(* PLC project liner_cyclic.project, CODESYS CODESYS V3.5 SP17 Patch 3 *)
(* stored: creationDateTime 1970-01-01T00:00:00, modificationDateTime 1970-01-01T00:00:00 *)

{attribute 'qualified_only'}
VAR_GLOBAL  (* GVL *)
  PDI0_CON_24V_ST : BOOL;  (* ////////DI//////////// /////////A11_ICPDAS_ECAT2053_v2//////////////////////// *)
  PDI1_SAFE_A_ST : BOOL;  (* Реле безопасности #1 *)
  PDI2_SAFE_B_ST : BOOL;  (* Реле безопасности #2 *)
  PDI3_CON_220V_ST : BOOL;  (* Цепи управления 220V, вентиляция шкафа, вентиляторы на моторах *)
  PDI4_UPS_24V_ST : BOOL;  (* Сигнал от ИБП - выходное напряжение ОК *)
  PDI5_UPS_ACCU_FL_bad : BOOL;  (* Сигнал от ИБП - аккумулятор плохой *)
  PDI6_UPS_ACCU_FL_wrk : BOOL;  (* Сигнал от ИБП - работа от аккумулятора *)
  PDI7_F1_LS_UP : BOOL;  (* Аварийный КВ крайнее положение (Верх) *)
  PDI8_F1_LS_DN : BOOL;  (* Аварийный КВ крайнее положение (Низ) *)
  PDI9_F1_LS_BP : BOOL;  (* Снятие с концевика вертикальный силовозб. *)
  PDI10_F1_PWR_ST : BOOL;  (* Силовой контактор *)
  PDI11_F1_FAN_ST : BOOL;  (* Вентилятор включен *)
  PDI12_F1_T_ST : BOOL;  (* Температура двигателя в норме *)
  PDI13_LS_DOOR_left : BOOL;  (* КВ "Дверь открыта левая" *)
  PDI14_LS_DOOR2_right : BOOL;  (* КВ "Дверь 2 открыта правая" *)
  PDQ0_COL_24V : BOOL;  (* /////////DO/////////////// /////////A13_ICPDAS_ECAT2057P//////////////////////// *)
  PDQ1_COL_RD : BOOL;  (* Светосигнальная колонна - красный *)
  PDQ2_COL_GN : BOOL;  (* Светосигнальная колонна - зелёный *)
  PDQ3_COL_SN : BOOL;  (* Светосигнальная колонна - зуммер *)
  PDQ4_F1_PWR_OO : BOOL;  (* Силовое питание -линейный силовозбудит. *)
  PDQ5_F1_LS_BYP : BOOL;  (* Ключ для снятия с концевиков *)
  PDQ6_F1_FAN_OO : BOOL;  (* Вентилятор вкл/выкл *)
  PAI_F1_FORCE_A5 : INT;  (* ////////AI//////////////// /////////A14_ICPDAS_ECAT2016N//////////////////////// *)
  ECAT2016N_Status_Underrange : BOOL;  (* ///////////////////////A14_ICPDAS_ECAT2016N СТАТУСЫ////////////////////////////// *)
  ECAT2016N_Status_Overrange : BOOL;
  ECAT2016N_Status_Limit_1_1 : BOOL;
  ECAT2016N_Status_Limit_1_2 : BOOL;
  ECAT2016N_Status_Limit_2_1 : BOOL;
  ECAT2016N_Status_Limit_2_2 : BOOL;
  ECAT2016N_Status_Error : BOOL;
  ECAT2016N_Status_TxPDO_State : BOOL;
  ECAT2016N_Status_TxPDO_Toggle : BOOL;
  KTSL_Status_1 : UINT;  (* ////////////////////KTSL_L1000///////////////////////////////// *)
  KTSL_Position_1 : UDINT;
  KTSL_Velocity_1 : DINT;
  Control_Word_out : UINT;  (* ////////////////////Veichi SD700///////////////////////////////// *)
  Target_Position_out : DINT;
  Target_Velocity_out : DINT;
  Status_Word_in : UINT;
  Actual_Position_in : DINT;
  Velocity_actual_value_in : DINT;
  GVLlrMoveAbsolutePosition : LREAL;  (* ////////////////////////////////////////////////////////////////// *)
  bAlarm : BOOL;
  breset_btn : BOOL;
  bfbJogJogForward : BOOL;
  bfbJogJogBackward : BOOL;
  bfbFollowVelocityOn : BOOL;
  bMainDelay : BOOL;
END_VAR
